{region '#Template'}
	{attribute 'Version' := '0.0.1.0'}
	{attribute 'Tags' := '"LCID": "1031", "Text": "Universal, Control, Event classes, Notification"'}
	{attribute 'Tags' := '"LCID": "1033", "Text": "Universal, Control, Event classes, Notification"'}
	{attribute 'Description' := '"LCID": "1031", "Text": "Ereignisklasse"'}
	{attribute 'Description' := '"LCID": "1033", "Text": "Event classes"'}
{endregion}
FUNCTION_BLOCK FB_BA_EvtCategory_SimpStandExt EXTENDS FB_BA_View
VAR_INPUT CONSTANT
	Simple				: FB_BA_EC;  
	Standard			: FB_BA_EC;
	Extended			: FB_BA_EC;
END_VAR

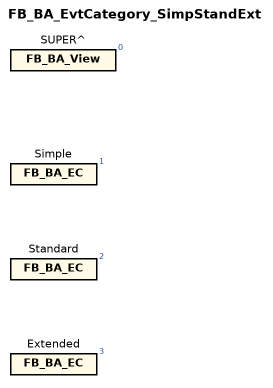
SUPER^(); // FB_BA_View
Simple(); // FB_BA_EC
Standard(); // FB_BA_EC
Extended(); // FB_BA_EC

METHOD FB_init : BOOL
VAR_INPUT
	bInitRetains : BOOL; // if TRUE, the retain variables are initialized (warm start / cold start)
	bInCopyCode : BOOL;  // if TRUE, the instance afterwards gets moved into the copy code (online change)
END_VAR
Simple.iParent					:= THIS^;
Simple.iLabel					:= LblControl.EvtClassSimple;									  
Simple.nInstanceID				:= EventClasses.LifeSafetySimple;
Simple.sObjectName				:= '{Idx=12}';
Simple.eEventType				:= E_BA_EventType.eAlarm;
Simple.eAlarmMode				:= E_BA_AlarmMode.eSimple;
Simple.aPriority[1]				:= 10;
Simple.aPriority[2]				:= 11;
Simple.aPriority[3]				:= 12;

Standard.iParent				:= THIS^;
Standard.iLabel					:= LblControl.EvtClassStandard;
Standard.nInstanceID			:= EventClasses.LifeSafetyStandard;
Standard.sObjectName			:= '{Idx=11}';
Standard.eEventType				:= E_BA_EventType.eAlarm;
Standard.eAlarmMode				:= E_BA_AlarmMode.eStandard;
Standard.aPriority[1]			:= 13;
Standard.aPriority[2]			:= 14;
Standard.aPriority[3]			:= 15;

Extended.iParent				:= THIS^;
Extended.iLabel					:= LblControl.EvtClassExtended;
Extended.nInstanceID			:= EventClasses.LifeSafetyExtended;
Extended.sObjectName			:= '{Idx=10}';
Extended.eEventType				:= E_BA_EventType.eAlarm;
Extended.eAlarmMode				:= E_BA_AlarmMode.eExtended;
Extended.aPriority[1]			:= 16;
Extended.aPriority[2]			:= 17;
Extended.aPriority[3]			:= 18;
END_METHOD

END_FUNCTION_BLOCK

(* stored: Version 1.1.0.1, ProductVersion 3.1.4024.6
   POU FB_BA_EvtCategory_SimpStandExt: Id {ab3da8b1-539b-416f-a65e-d45ed561d35e}, SpecialFunc None
   Method FB_init: Id {3b5c2880-11ac-45b9-ab1f-68d2ec623904} *)
